FUNCTION_BLOCK L3_MachineChecker (* Basic Function Block Type *)
  (* Standard: 61499-2 *)
  (* Version 0.0, 2014-11-06, EQUEROL, UJI *)
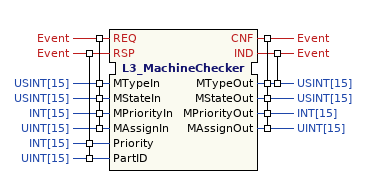
  EVENT_INPUT
    REQ WITH MTypeIn, MStateIn, MPriorityIn, MAssignIn; (* Normal Execution Request *)
    RSP WITH Priority, PartID; (* Response from PPTable *)
  END_EVENT
  EVENT_OUTPUT
    CNF WITH MTypeOut, MStateOut, MPriorityOut, MAssignOut; (* Execution Confirmation *)
    IND WITH MTypeOut; (* Indication to the process plan table *)
  END_EVENT
  VAR_INPUT
    MTypeIn : ARRAY [0..14] OF USINT; (* Machine type vector *)
    MStateIn : ARRAY [0..14] OF USINT; (* Machine state vector *)
    MPriorityIn : ARRAY [0..14] OF INT; (* Machine priorities vector *)
    MAssignIn : ARRAY [0..14] OF UINT; (* Machine assignation vector *)
    Priority : ARRAY [0..14] OF INT; (* PP priorities vector *)
    PartID : ARRAY [0..14] OF UINT; (* Part identifiers vector *)
  END_VAR
  VAR_OUTPUT
    MTypeOut : ARRAY [0..14] OF USINT; (* Machine type vector *)
    MStateOut : ARRAY [0..14] OF USINT; (* MAchine state vector *)
    MPriorityOut : ARRAY [0..14] OF INT; (* Machine priorities vector *)
    MAssignOut : ARRAY [0..14] OF UINT; (* Machine assignation vector *)
  END_VAR
  VAR
    i : USINT := 0; (* loop variable *)
  END_VAR
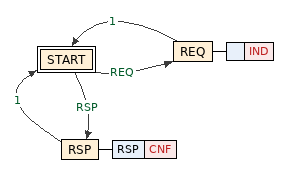
  EC_STATES
    START; (* Initial State *)
    REQ : -> IND; (* Normal execution *)
    RSP : RSP -> CNF;
  END_STATES
  EC_TRANSITIONS
    START TO REQ := REQ;
    REQ TO START := 1;
    START TO RSP := RSP;
    RSP TO START := 1;
  END_TRANSITIONS
  ALGORITHM RSP IN ST: (* Response from PPTable algorithm *)
FOR i := 0 TO 14 DO
	MTypeOut[i] := MTypeIn[i];
	MStateOut[i] := MStateIn[i];
	MPriorityOut[i] := MPriorityIn[i];
	MAssignOut[i] := MAssignIn[i];

	IF MStateIn[i] = 2 THEN
	(*Temp fix #, only take machines that are free and ready*)
		IF Priority[i] < MPriorityIn[i] THEN
			(*1st to get into the vector has preference when prios are equal*)
			MPriorityOut[i] := Priority[i];
			MAssignOut[i] := PartID[i];
		END_IF;
	END_IF;
END_FOR;
  END_ALGORITHM
END_FUNCTION_BLOCK
